FUNCTION_BLOCK PIOC_Logic (* Basic Function Block Type *)
  (* Standard: 61499-2 *)
  (* Version 0.0, 12/10/2023, Cheyan, Schneider Electric, Template *)
  PACKAGE Main;
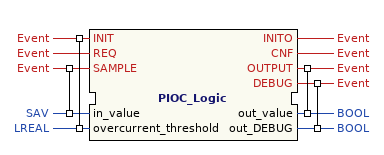
  EVENT_INPUT
    INIT WITH overcurrent_threshold; (* Initialization Request *)
    REQ; (* Normal Execution Request *)
    SAMPLE WITH in_value;
  END_EVENT
  EVENT_OUTPUT
    INITO; (* Initialization Confirm *)
    CNF; (* Execution Confirmation *)
    OUTPUT WITH out_value;
    DEBUG WITH out_DEBUG;
  END_EVENT
  VAR_INPUT
    in_value : SAV; (* Input event qualifier *)
    overcurrent_threshold : LREAL;
  END_VAR
  VAR_OUTPUT
    out_value : BOOL;
    out_DEBUG : BOOL;
  END_VAR
  VAR
    overcurrent_counter_internal : DINT := 0;
  END_VAR
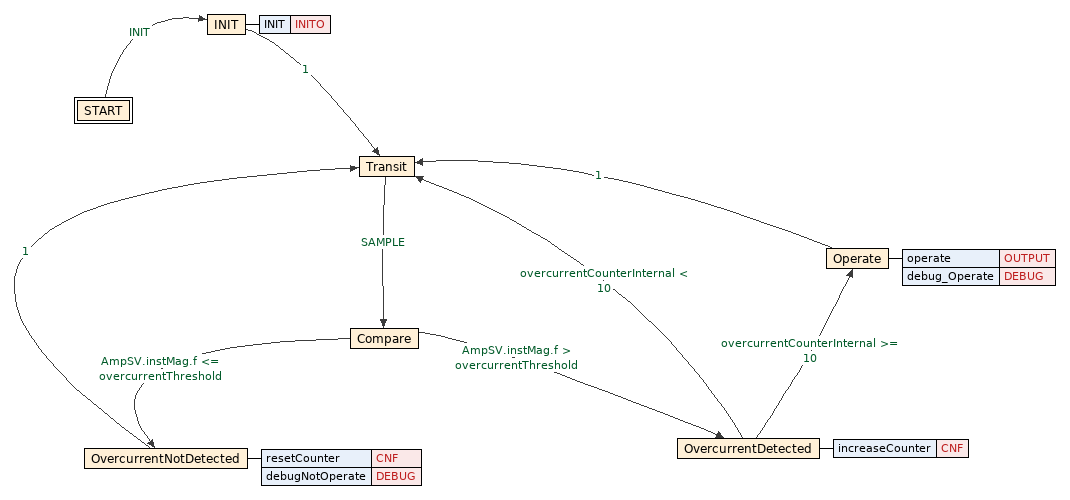
  EC_STATES
    START; (* Initial State *)
    INIT : INIT -> INITO; (* Initialization *)
    Transit; (* Normal execution *)
    OvercurrentNotDetected : resetCounter -> CNF, debugNotOperate -> DEBUG;
    OvercurrentDetected : increaseCounter -> CNF;
    Compare;
    Operate : operate -> OUTPUT, debug_Operate -> DEBUG;
  END_STATES
  EC_TRANSITIONS
    START TO INIT := INIT;
    INIT TO Transit := 1;
    Compare TO OvercurrentNotDetected := AmpSV.instMag.f <= overcurrentThreshold;
    Compare TO OvercurrentDetected := AmpSV.instMag.f > overcurrentThreshold;
    Transit TO Compare := SAMPLE;
    OvercurrentNotDetected TO Transit := 1;
    OvercurrentDetected TO Operate := overcurrentCounterInternal >= 10;
    Operate TO Transit := 1;
    OvercurrentDetected TO Transit := overcurrentCounterInternal < 10;
  END_TRANSITIONS
  ALGORITHM INIT IN ST: (* Initialization algorithm *)
;
  END_ALGORITHM
  ALGORITHM resetCounter IN ST: (* Set the overcurrent counter to 0 *)
;

overcurrent_counter_internal := 0;
  END_ALGORITHM
  ALGORITHM increaseCounter IN ST: (* increase the internal overcurrent counter *)
;

overcurrent_counter_internal := overcurrent_counter_internal + 1;
  END_ALGORITHM
  ALGORITHM operate IN ST: (* When an overcurrent fault is detected (after detection of 10 overcurrent measurement), Op_general is set to FALSE *)
;

out_value := TRUE;
  END_ALGORITHM
  ALGORITHM notOperate IN ST:
;

out_value := FALSE;
  END_ALGORITHM
  ALGORITHM debug_Operate IN ST:
;

out_DEBUG := TRUE;
  END_ALGORITHM
  ALGORITHM debugNotOperate IN ST:
;

out_DEBUG := FALSE;
  END_ALGORITHM
END_FUNCTION_BLOCK
